TYPE "UDT_main"
TITLE = Datatype Main
VERSION : 0.1
//here is the comment
   STRUCT
      one : Bool;   // comment one
      two {InstructionName := 'DTL'; LibVersion := '1.0'} : Array[0..10] of DTL;   // comment two
      three : Byte;   // comment three
      four : Word;   // comment four
      five : DWord;   // comment five
      aa_comment_free : "UDT_commentfree";   // comment aa_comment_free
      ab_with_subudt : "UDT with sub udt";   // comment UDT with subudt
      ac_without_subudt : "UDT_without_sub_udt";   // comment UDT without subudt
      six : Word;   // comment six
      seven : SInt;   // comment seven
      eight : USInt;   // comment eight
      multiarray_01 : Array[0..5, 0..2, 1..3] of Bool;   // comment multiarray_01
      multiarray_02 : Array[0..5, 0..1] of Byte;   // comment multiarray_02
      multiarray_03 : Array[0..2, 0..1] of "UDT_without_sub_udt";   // comment multiarray_03
      nine : Int;   // comment nine
      ten : UInt;   // comment ten
      eleven : DInt;   // comment eleven
      twelve : UDInt;   // comment twelve
      thirteen : Int;   // comment thirteen
      fourteen : Int;   // comment fourteen
      fifteen : Real;   // comment fifteen
      sixteenn : LReal;   // comment sixteen
      seventeen : Char;   // comment seventeen
      eighteen : WChar;   // comment eighteen
      nineteen : String;   // comment nineteen
      twenty : WString;   // comment twenty
      twentyone {InstructionName := 'DTL'; LibVersion := '1.0'} : DTL;   // comment twentyone
      twentytwo : Array[0..10] of Byte;   // comment twentytwo
      twentythree : Struct   // // comment twentythree
         A : Bool;   // comment A
         B : Int;   // comment B
         C : "UDT_without_sub_udt";   // comment C
         D : "UDT_without_sub_udt";   // comment D
         E : DInt;   // comment E
      END_STRUCT;
      twentysix : Bool;   // comment twentysix
   END_STRUCT;

END_TYPE

